Staubli VAL3: decodePose.pgx

program decodePose(joint& value, num& buffer[])
  local num decodeBuffer[6]
begin
  fromBinary(buffer, 24, "4.0b", decodeBuffer)

  value = {decodeBuffer[0], decodeBuffer[1], decodeBuffer[2], decodeBuffer[3], decodeBuffer[4], decodeBuffer[5]}

  logMsg("J: (" + toString("3", value.j1) + ", " + toString("3", value.j2) + ", " + toString("3", value.j3) + ", " + toString("3", value.j4) + ", " + toString("3", value.j5) + ", " + toString("3", value.j6) + ")")
end
